// TIA Portal project "Refill_Work" (V19)

(* hardware
DEVICE "S7-1500/ET200MP station_1"  S7-1500 station
   slot 0: "Rail_0"  Rack  6ES7 590-1***0-0AA0
   slot 1: "PLC_Refil_Work"  CPU 1511-1 PN  6ES7 511-1AK01-0AB0  V2.9
      slot 3: "CPU display_1"  6ES7591-1AA00-0AA0
      slot 32768: "PROFINET interface_1"  X1
         slot 32769: "Port_1"  X1 P1
         slot 32770: "Port_2"  X1 P2
      slot 34817: "Virtual CP interface port_1"  Virtual CP interface port  Virtual CP interface port
   slot 2: "DI 16x24VDC BA_1"  DI 16x24VDC BA  6ES7 521-1BH10-0AA0  V1.1
   slot 3: "DQ 16x24VDC/0.5A BA_1"  DQ 16x24VDC/0.5A BA  6ES7 522-1BH10-0AA0  V1.1
   slot 4: "AI 4xU/I/RTD/TC ST_1"  AI 4xU/I/RTD/TC ST  6ES7 531-7QD00-0AB0  V1.0
*)

// ===== PLC "PLC_Refil_Work"  CPU 1511-1 PN =====

VAR_GLOBAL   // PLC tag table "Default tag table"
   "System_Byte" AT %MB1 : Byte;
   "FirstScan" AT %M1.0 : Bool;
   "DiagStatusUpdate" AT %M1.1 : Bool;
   "AlwaysTRUE" AT %M1.2 : Bool;
   "AlwaysFALSE" AT %M1.3 : Bool;
   "Clock_Byte" AT %MB0 : Byte;
   "Clock_10Hz" AT %M0.0 : Bool;
   "Clock_5Hz" AT %M0.1 : Bool;
   "Clock_2.5Hz" AT %M0.2 : Bool;
   "Clock_2Hz" AT %M0.3 : Bool;
   "Clock_1.25Hz" AT %M0.4 : Bool;
   "Clock_1Hz" AT %M0.5 : Bool;
   "Clock_0.625Hz" AT %M0.6 : Bool;
   "Clock_0.5Hz" AT %M0.7 : Bool;
END_VAR

VAR_GLOBAL   // PLC tag table "Outputs Machine"
   "q_xLamp_Running" AT %Q2.0 : Bool;
   "q_xLamp_Faulted" AT %Q2.1 : Bool;
END_VAR

VAR_GLOBAL   // PLC tag table "Inputs Machine"
   "i_xButton_Start" AT %I0.0 : Bool;
   "i_xButton_Stop" AT %I0.1 : Bool;
   "i-xButton_Reset" AT %I0.2 : Bool;
END_VAR

VAR_GLOBAL   // PLC tag table "Outputs Equipment"
   "q_xRefill_Pump_Start_P1" AT %Q3.0 : Bool;
   "q_xRefill_Valve_Open_P1" AT %Q3.1 : Bool;
   "q_xRefill_Pump_Start_P2" AT %Q3.2 : Bool;
   "q_xRefill_Valve_Open_P2" AT %Q3.3 : Bool;
END_VAR

VAR_GLOBAL   // PLC tag table "Inputs Equipment"
   "i_xRefill_Pump_MCB_P1" AT %I0.3 : Bool;
   "i_xRefill_Pump_LI_P1" AT %I0.4 : Bool;
   "i_xRefill_Pump_Running_P1" AT %I0.5 : Bool;
   "i_xRefill_Valve_Open_P1" AT %I0.6 : Bool;
   "i_iRefill_Tank_ActLevel_p1" AT %IW4 : Int;
   "I_xRefill_Pump_MCB_P2" AT %I0.7 : Bool;
   "i_xRefill_Pump_LI_P2" AT %I1.0 : Bool;
   "i_xRefill_PumpRunning_P2" AT %I1.1 : Bool;
   "i_xRefill_Valve_Open_P2" AT %I1.2 : Bool;
   "i_iRefill_Tank_ActLevel_P2" AT %IW6 : Int;
   "i_xSupply_Tank_LowLever" AT %I1.3 : Bool;
END_VAR

TYPE "UDT_Statehandler"
   STRUCT
      State : Struct
         xReady : Bool;
         xRunning : Bool;
         xFaulted : Bool;
         xReset : Bool;
      END_STRUCT;
      Cmd : Struct
         xStart : Bool;
         xStop : Bool;
         xReset : Bool;
      END_STRUCT;
   END_STRUCT;
END_TYPE

TYPE "UDT_Supply"
   STRUCT
      Status : Struct
         xLowLever : Bool;
         xFaulted : Bool;
      END_STRUCT;
      Cmd : Struct
         xSpare : Bool;
      END_STRUCT;
      Cfg : Struct
         xSpare : Bool;
      END_STRUCT;
      Fit : Struct
         wTrigger : Word;
      END_STRUCT;
   END_STRUCT;
END_TYPE

// folder: Equipment

TYPE "UDT_Refill"
   STRUCT
      Status : Struct
         iLevel : Int;
         xPumpRunning : Bool;
         xFaulted : Bool;
      END_STRUCT;
      Cmd : Struct
         xRequestRefill : Bool;
      END_STRUCT;
      Cfg : Struct
         xSpare : Bool;
      END_STRUCT;
      Fit : Struct
         wTrigger : Word;
      END_STRUCT;
   END_STRUCT;
END_TYPE

// folder: 00Machine

DATA_BLOCK "Instance Machine Modules"   // DB1
{ S7_Optimized_Access := 'TRUE' }
VERSION : 0.1
// stored: InstanceOfName FB - Machine Modules
"FB - Machine Modules"
BEGIN
END_DATA_BLOCK

// folder: 01Equipment

DATA_BLOCK "Inctance Equipment Modules"   // DB2
{ S7_Optimized_Access := 'TRUE' }
VERSION : 0.1
// stored: InstanceOfName FB - Equipment Modules
"FB - Equipment Modules"
BEGIN
END_DATA_BLOCK

// folder: 02GlobalData

DATA_BLOCK "DB - Machine"   // DB3
{ S7_Optimized_Access := 'TRUE' }
VERSION : 0.1
   VAR
      Statehandler : "UDT_Statehandler";
   END_VAR
BEGIN
END_DATA_BLOCK

DATA_BLOCK "DB - Equipment"   // DB3
{ S7_Optimized_Access := 'TRUE' }
VERSION : 0.1
   VAR
      Supply : "UDT_Supply";
      Refil_Process_1 : "UDT_Refill";
      Refil_Process_2 : "UDT_Refill";
   END_VAR
BEGIN
END_DATA_BLOCK

// folder: (top level)

ORGANIZATION_BLOCK "Main"   // OB1, LAD, ProgramCycle
TITLE = "Main Program Sweep (Cycle)"
{ S7_Optimized_Access := 'TRUE' }
VERSION : 0.1
   VAR_INPUT
      Initial_Call : Bool;   // Initial call of this OB
      Remanence : Bool;   // =True, if remanent data are available
   END_VAR
BEGIN

REGION Network 1: Call - Main machine modules
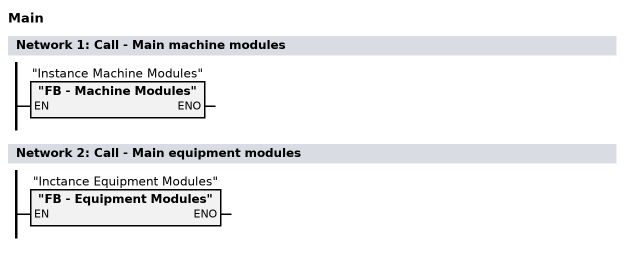
   RUNG wire#powerrail
      "Instance Machine Modules"()
   END_RUNG
   // the same network as SCL:
   "Instance Machine Modules"();   // "FB - Machine Modules"
END_REGION

REGION Network 2: Call - Main equipment modules
   RUNG wire#powerrail
      "Inctance Equipment Modules"()
   END_RUNG
   // the same network as SCL:
   "Inctance Equipment Modules"();   // "FB - Equipment Modules"
END_REGION
END_ORGANIZATION_BLOCK

// folder: 00Machine

FUNCTION_BLOCK "FB - Machine Modules"   // FB1, LAD
TITLE = FB - Machine Calls
{ S7_Optimized_Access := 'TRUE' }
VERSION : 0.1
   VAR
      Instance_StateHandler : "FB - StateHandler";
   END_VAR
   VAR_TEMP
      _info : Struct
         xReady : Bool;
         xRunning : Bool;
         xFaulted : Bool;
         xReset : Bool;
      END_STRUCT;
   END_VAR
BEGIN

REGION Network 1: MODULE - State Handler
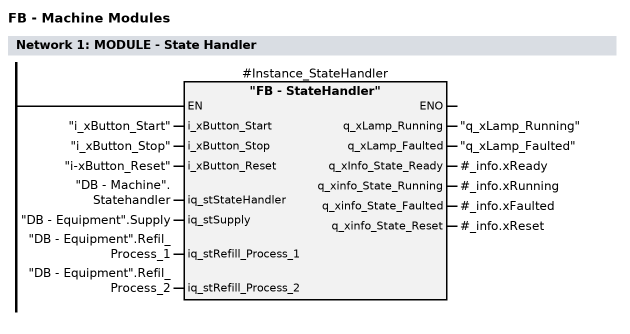
   RUNG wire#powerrail
      #Instance_StateHandler(i_xButton_Start := "i_xButton_Start", i_xButton_Stop := "i_xButton_Stop", i_xButton_Reset := "i-xButton_Reset", iq_stStateHandler := "DB - Machine".Statehandler, iq_stSupply := "DB - Equipment".Supply, iq_stRefill_Process_1 := "DB - Equipment".Refil_Process_1, iq_stRefill_Process_2 := "DB - Equipment".Refil_Process_2, q_xLamp_Running => "q_xLamp_Running", q_xLamp_Faulted => "q_xLamp_Faulted", q_xInfo_State_Ready => #_info.xReady, q_xinfo_State_Running => #_info.xRunning, q_xinfo_State_Faulted => #_info.xFaulted, q_xinfo_State_Reset => #_info.xReset)
   END_RUNG
   // the same network as SCL:
   #Instance_StateHandler(i_xButton_Start := "i_xButton_Start",   // "FB - StateHandler"
                          i_xButton_Stop := "i_xButton_Stop",
                          i_xButton_Reset := "i-xButton_Reset",
                          iq_stStateHandler := "DB - Machine".Statehandler,
                          iq_stSupply := "DB - Equipment".Supply,
                          iq_stRefill_Process_1 := "DB - Equipment".Refil_Process_1,
                          iq_stRefill_Process_2 := "DB - Equipment".Refil_Process_2,
                          q_xLamp_Running => "q_xLamp_Running",
                          q_xLamp_Faulted => "q_xLamp_Faulted",
                          q_xInfo_State_Ready => #_info.xReady,
                          q_xinfo_State_Running => #_info.xRunning,
                          q_xinfo_State_Faulted => #_info.xFaulted,
                          q_xinfo_State_Reset => #_info.xReset);
END_REGION
END_FUNCTION_BLOCK

// folder: 00Machine/Functions

FUNCTION_BLOCK "FB - StateHandler"   // FB2, LAD
TITLE = MACHINE - State Handler
{ S7_Optimized_Access := 'TRUE' }
VERSION : 0.1
   VAR_INPUT
      i_xButton_Start : Bool;
      i_xButton_Stop : Bool;
      i_xButton_Reset : Bool;
   END_VAR
   VAR_OUTPUT
      q_xLamp_Running : Bool;
      q_xLamp_Faulted : Bool;
      q_xInfo_State_Ready : Bool;
      q_xinfo_State_Running : Bool;
      q_xinfo_State_Faulted : Bool;
      q_xinfo_State_Reset : Bool;
   END_VAR
   VAR_IN_OUT
      iq_stStateHandler : "UDT_Statehandler";
      iq_stSupply : "UDT_Supply";
      iq_stRefill_Process_1 : "UDT_Refill";
      iq_stRefill_Process_2 : "UDT_Refill";
   END_VAR
   VAR
      iState : Int;
      stOnDelay_Reset : TON_TIME;
   END_VAR
BEGIN

REGION Network 1: CONTROL - Start Operation
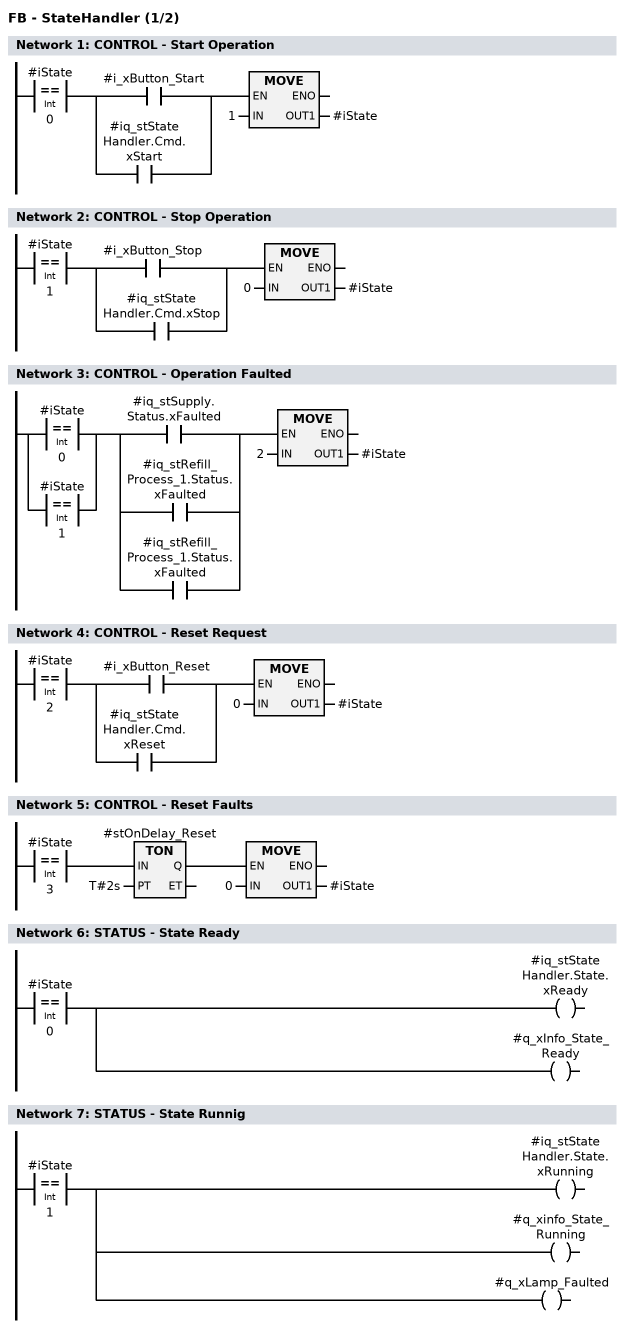
   RUNG wire#powerrail
      { S7_Templates := "SrcType := Int" } EQ_Contact(in1 := #iState, in2 := 0)
      wire#w1
      Contact( #i_xButton_Start )
      wire#w2
      Move(in := 1, out1 => #iState)
   END_RUNG
   RUNG wire#w1
      Contact( #iq_stStateHandler.Cmd.xStart )
   END_RUNG wire#w2
   // the same network as SCL:
   IF (#iState = 0) AND (#i_xButton_Start OR #iq_stStateHandler.Cmd.xStart) THEN #iState := 1; END_IF;
END_REGION

REGION Network 2: CONTROL - Stop Operation
   RUNG wire#powerrail
      { S7_Templates := "SrcType := Int" } EQ_Contact(in1 := #iState, in2 := 1)
      wire#w1
      Contact( #i_xButton_Stop )
      wire#w2
      Move(in := 0, out1 => #iState)
   END_RUNG
   RUNG wire#w1
      Contact( #iq_stStateHandler.Cmd.xStop )
   END_RUNG wire#w2
   // the same network as SCL:
   IF (#iState = 1) AND (#i_xButton_Stop OR #iq_stStateHandler.Cmd.xStop) THEN #iState := 0; END_IF;
END_REGION

REGION Network 3: CONTROL - Operation Faulted
   RUNG wire#powerrail
      { S7_Templates := "SrcType := Int" } EQ_Contact(in1 := #iState, in2 := 0)
      wire#w1
      Contact( #iq_stSupply.Status.xFaulted )
      wire#w2
      Move(in := 2, out1 => #iState)
   END_RUNG
   RUNG wire#powerrail
      { S7_Templates := "SrcType := Int" } EQ_Contact(in1 := #iState, in2 := 1)
   END_RUNG wire#w1
   RUNG wire#w1
      Contact( #iq_stRefill_Process_1.Status.xFaulted )
   END_RUNG wire#w2
   RUNG wire#w1
      Contact( #iq_stRefill_Process_1.Status.xFaulted )
   END_RUNG wire#w2
   // the same network as SCL:
   IF ((#iState = 0) OR (#iState = 1)) AND (#iq_stSupply.Status.xFaulted OR #iq_stRefill_Process_1.Status.xFaulted OR #iq_stRefill_Process_1.Status.xFaulted) THEN
       #iState := 2;
   END_IF;
END_REGION

REGION Network 4: CONTROL - Reset Request
   RUNG wire#powerrail
      { S7_Templates := "SrcType := Int" } EQ_Contact(in1 := #iState, in2 := 2)
      wire#w1
      Contact( #i_xButton_Reset )
      wire#w2
      Move(in := 0, out1 => #iState)
   END_RUNG
   RUNG wire#w1
      Contact( #iq_stStateHandler.Cmd.xReset )
   END_RUNG wire#w2
   // the same network as SCL:
   IF (#iState = 2) AND (#i_xButton_Reset OR #iq_stStateHandler.Cmd.xReset) THEN #iState := 0; END_IF;
END_REGION

REGION Network 5: CONTROL - Reset Faults
   #stOnDelay_Reset(IN := #iState = 3, PT := T#2s);   // TON
   IF #stOnDelay_Reset.Q THEN #iState := 0; END_IF;
END_REGION

REGION Network 6: STATUS - State Ready
   RUNG wire#powerrail
      { S7_Templates := "SrcType := Int" } EQ_Contact(in1 := #iState, in2 := 0)
      wire#w1
      Coil( #iq_stStateHandler.State.xReady )
   END_RUNG
   RUNG wire#w1
      Coil( #q_xInfo_State_Ready )
   END_RUNG
   // the same network as SCL:
   #iq_stStateHandler.State.xReady := #iState = 0;
   #q_xInfo_State_Ready := #iq_stStateHandler.State.xReady;
END_REGION

REGION Network 7: STATUS - State Runnig
   RUNG wire#powerrail
      { S7_Templates := "SrcType := Int" } EQ_Contact(in1 := #iState, in2 := 1)
      wire#w1
      Coil( #iq_stStateHandler.State.xRunning )
   END_RUNG
   RUNG wire#w1
      Coil( #q_xinfo_State_Running )
   END_RUNG
   RUNG wire#w1
      Coil( #q_xLamp_Faulted )
   END_RUNG
   // the same network as SCL:
   #iq_stStateHandler.State.xRunning := #iState = 1;
   #q_xinfo_State_Running := #iq_stStateHandler.State.xRunning;
   #q_xLamp_Faulted := #iq_stStateHandler.State.xRunning;
END_REGION

REGION Network 8: STATUS - State Faulted
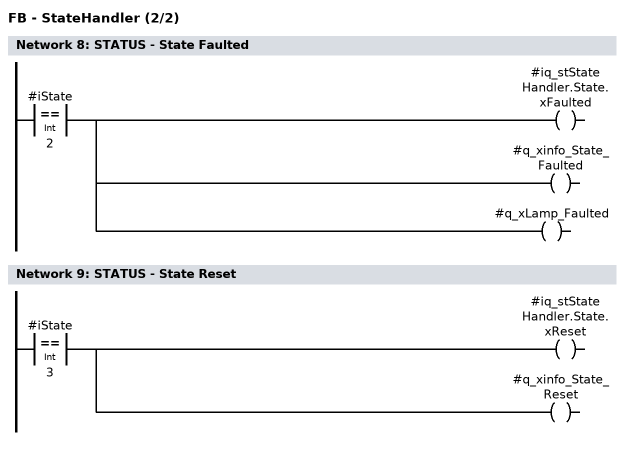
   RUNG wire#powerrail
      { S7_Templates := "SrcType := Int" } EQ_Contact(in1 := #iState, in2 := 2)
      wire#w1
      Coil( #iq_stStateHandler.State.xFaulted )
   END_RUNG
   RUNG wire#w1
      Coil( #q_xinfo_State_Faulted )
   END_RUNG
   RUNG wire#w1
      Coil( #q_xLamp_Faulted )
   END_RUNG
   // the same network as SCL:
   #iq_stStateHandler.State.xFaulted := #iState = 2;
   #q_xinfo_State_Faulted := #iq_stStateHandler.State.xFaulted;
   #q_xLamp_Faulted := #iq_stStateHandler.State.xFaulted;
END_REGION

REGION Network 9: STATUS - State Reset
   RUNG wire#powerrail
      { S7_Templates := "SrcType := Int" } EQ_Contact(in1 := #iState, in2 := 3)
      wire#w1
      Coil( #iq_stStateHandler.State.xReset )
   END_RUNG
   RUNG wire#w1
      Coil( #q_xinfo_State_Reset )
   END_RUNG
   // the same network as SCL:
   #iq_stStateHandler.State.xReset := #iState = 3;
   #q_xinfo_State_Reset := #iq_stStateHandler.State.xReset;
END_REGION
END_FUNCTION_BLOCK

// folder: 01Equipment

FUNCTION_BLOCK "FB - Equipment Modules"   // FB1, LAD
{ S7_Optimized_Access := 'TRUE' }
VERSION : 0.1
BEGIN
END_FUNCTION_BLOCK